Staubli VAL3: onF7Event.pgx

program onF7Event()
  local num l_nIndex
  local string l_sItem
  local num i
  local num l_nResult
  local string l_sMessage
begin
  // look if the bButton is enable
  if bButton[6]
    //
  endIf
end
